(*8.计数器清零*)	
	IF GVL_State.iPLC_State=50 THEN
		(*-----------------------计数器清零操作-----------------------*)
		IF PLC_PRG.Step_Scout<=42 OR PLC_PRG.Step_Scout>=70 THEN
			iActNumPulse:=0;
			Entity_IO.bTriggerOut:=FALSE;
			Entity_IO.bTriggerPannel_NOT:=FALSE;
		END_IF
	ELSIF GVL_State.iPLC_State=60 THEN
		(*-----------------------计数器清零操作-----------------------*)
		IF PLC_PRG.Step_CBCT<=70 THEN
			iActNumPulse:=0;
			Entity_IO.bTriggerOut:=FALSE;
			Entity_IO.bTriggerPannel_NOT:=FALSE;
		END_IF
	ELSIF GVL_State.iPLC_State=40 THEN
		iActNumPulse:=0;
	END_IF

END_PROGRAM

// Device/Application/Motor
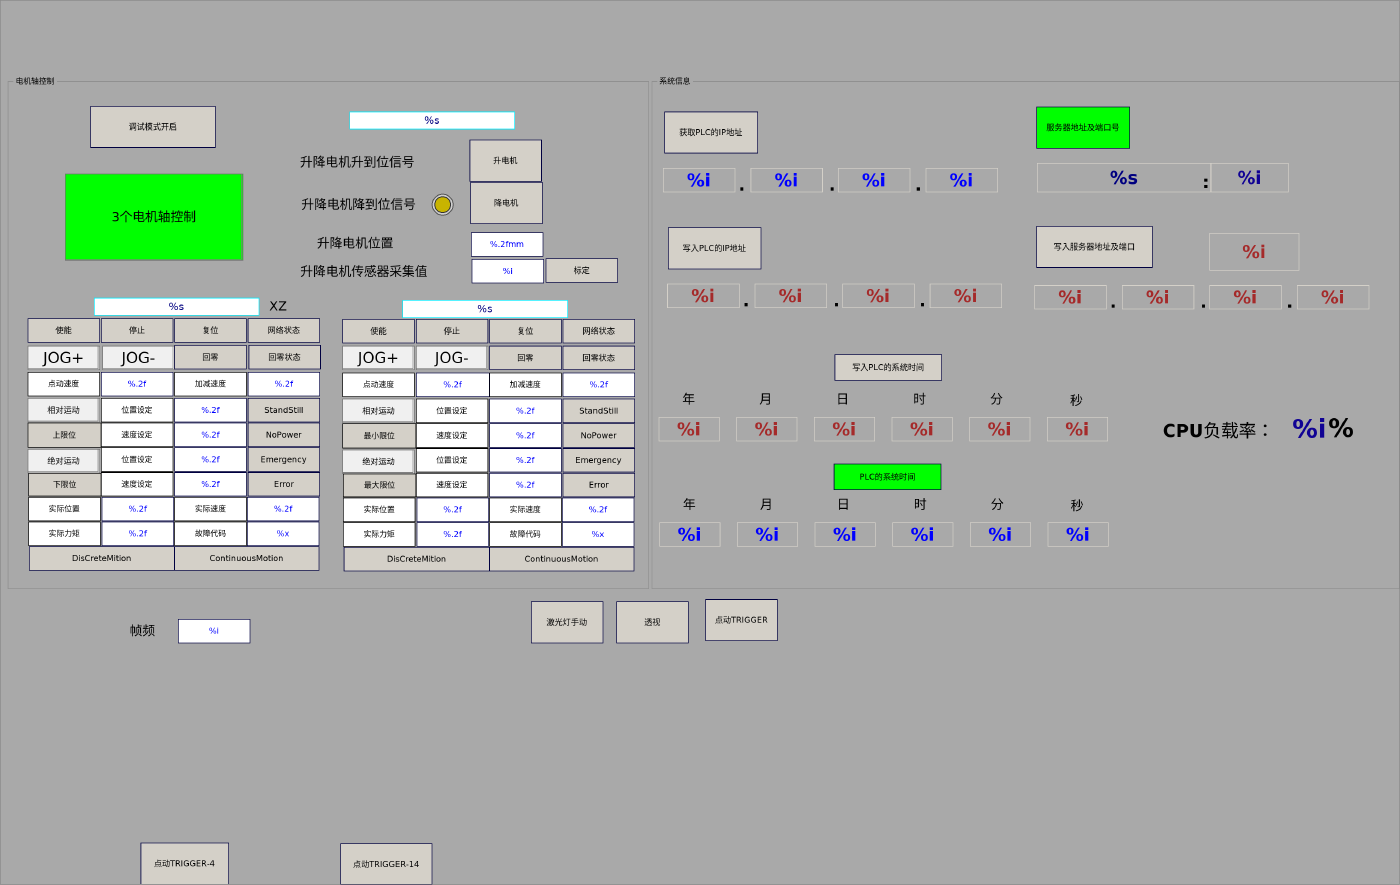
VISUALIZATION Motor  // 1983x1254
    Button (39,490 102x34), "JOG+", colour toggle: Axis_XZ.XZ_AxisCmd.bJogP
        tap Axis_XZ.XZ_AxisCmd.bJogP
    Rectangle (144,704 102x34), "%.2f", text variable: Axis_XZ.XZ_AxisState.rActPosition
    Button (145,490 102x34), "JOG-", colour toggle: Axis_XZ.XZ_AxisCmd.bJogN
        tap Axis_XZ.XZ_AxisCmd.bJogN
    RoundedRectangle (39,451 102x34), "使能", colour toggle: AXIS_XZ.XZ_AxisState.bPowering
        toggle Axis_XZ.XZ_AxisCmd.bPower
    RoundedRectangle (351,451 102x34), "网络状态", colour toggle: Axis_XZ.XZ_AxisState.bNetState
    Button (39,636 102x34), "绝对运动", colour toggle: Axis_XZ.XZ_AxisCmd.bAbs
        tap Axis_XZ.XZ_AxisCmd.bAbs
    Rectangle (40,704 102x34), "实际位置"
    Rectangle (350,704 102x34), "%.2f", text variable: Axis_XZ.XZ_AxisState.rActVelocity
    Rectangle (247,704 102x34), "实际速度"
    RoundedRectangle (143,451 102x34), "停止", colour toggle: Axis_XZ.XZ_AxisState.bStopState
        tap Axis_XZ.XZ_AxisCmd.bStop
    RoundedRectangle (247,451 102x34), "复位", colour toggle: Axis_XZ.XZ_AxisCmd.bReset
        tap Axis_XZ.XZ_AxisCmd.bReset
    Rectangle (133,422 234x25), "%s", text variable: InitMotor.sNameXZ, text list: ''
    Rectangle (247,739 102x34), "故障代码"
    Rectangle (350,739 102x34), "%x", text variable: Axis_XZ.XZ_AxisState.ErrorID, colour toggle: (Axis_XZ.XZ_AxisState.ErrorID)<>0
    Rectangle (40,670 103x33), "下限位", colour toggle: Entity_IO.bRotateMotorMax
    Rectangle (39,599 104x35), "上限位", colour toggle: Entity_IO.bRotateMotorMin
    RoundedRectangle (247,489 102x34), "回零", colour toggle: Axis_XZ.XZ_AxisCmd.bHome
        tap Axis_XZ.XZ_AxisCmd.bHome
    Button (39,564 102x34), "相对运动", colour toggle: Axis_XZ.XZ_AxisCmd.bRel
        tap Axis_XZ.XZ_AxisCmd.bRel
    Rectangle (143,527 102x34), "%.2f", text variable: Axis_XZ.XZ_AxisCmd.AxisPara.rJogVelocity
        OnMouseClick: write Axis_XZ.XZ_AxisCmd.AxisPara.rJogVelocity via Default
    Rectangle (39,527 102x34), "点动速度"
    Rectangle (247,527 102x34), "加减速度"
    Rectangle (351,527 102x34), "%.2f", text variable: Axis_XZ.XZ_AxisCmd.AxisPara.rAccDec
        OnMouseClick: write Axis_XZ.XZ_AxisCmd.AxisPara.rAccDec via Default
    Rectangle (143,564 102x34), "位置设定"
    Rectangle (247,564 102x34), "%.2f", text variable: Axis_XZ.XZ_AxisCmd.AxisPara.rRelPosition
        OnMouseClick: write Axis_XZ.XZ_AxisCmd.AxisPara.rRelPosition via Default
    Rectangle (143,599 102x34), "速度设定"
    Rectangle (247,599 102x34), "%.2f", text variable: Axis_XZ.XZ_AxisCmd.AxisPara.rRelVelocity
        OnMouseClick: write Axis_XZ.XZ_AxisCmd.AxisPara.rRelVelocity via Default
    Rectangle (143,634 102x34), "位置设定"
    Rectangle (693,635 102x34), "%.2f", text variable: Axis_QJ.QJ_AxisCmd.AxisPara.rAbsPosition
        OnMouseClick: write Axis_QJ.QJ_AxisCmd.AxisPara.rAbsPosition via Default
    Rectangle (143,669 102x34), "速度设定"
    Rectangle (247,669 102x34), "%.2f", text variable: Axis_XZ.XZ_AxisCmd.AxisPara.rAbsVelocity
        OnMouseClick: write Axis_XZ.XZ_AxisCmd.AxisPara.rAbsVelocity via Default
    RoundedRectangle (351,564 102x34), "StandStill", colour toggle: Axis_XZ.XZ_AxisState.bStandStill
    RoundedRectangle (351,599 102x34), "NoPower", colour toggle: Axis_XZ.XZ_AxisState.bPowerOff
    RoundedRectangle (351,634 102x34), "Emergency", colour toggle: Axis_XZ.XZ_AxisState.bErrStop
    RoundedRectangle (351,669 102x34), "Error", colour toggle: Axis_XZ.XZ_AxisState.bAxisErr
    Rectangle (144,739 102x34), "%.2f", text variable: Axis_XZ.XZ_AxisState.rActTorque
    Rectangle (40,739 102x34), "实际力矩"
    Rectangle (570,425 234x25), "%s", text variable: InitMotor.sNameQJ, text list: ''
    Button (485,490 102x34), "JOG+", colour toggle: Axis_QJ.QJ_AxisCmd.bJogP
        tap Axis_QJ.QJ_AxisCmd.bJogP
    Rectangle (590,705 102x34), "%.2f", text variable: Axis_QJ.QJ_AxisState.rActPosition
    Button (589,490 102x34), "JOG-", colour toggle: Axis_QJ.QJ_AxisCmd.bJogN
        tap Axis_QJ.QJ_AxisCmd.bJogN
    RoundedRectangle (485,452 102x34), "使能", colour toggle: AXIS_QJ.QJ_AxisState.bPowering
        toggle Axis_QJ.QJ_AxisCmd.bPower
    RoundedRectangle (797,452 102x34), "网络状态", colour toggle: Axis_QJ.QJ_AxisState.bNetState
    Button (485,637 102x34), "绝对运动", colour toggle: Axis_QJ.QJ_AxisCmd.bAbs
        tap Axis_QJ.QJ_AxisCmd.bAbs
    Rectangle (486,705 102x34), "实际位置"
    Rectangle (796,705 102x34), "%.2f", text variable: Axis_QJ.QJ_AxisState.rActVelocity
    Rectangle (693,705 102x34), "实际速度"
    RoundedRectangle (589,452 102x34), "停止", colour toggle: Axis_QJ.QJ_AxisCmd.bStop
        tap Axis_QJ.QJ_AxisCmd.bStop
    RoundedRectangle (693,452 102x34), "复位", colour toggle: Axis_QJ.QJ_AxisCmd.bReset
        tap Axis_QJ.QJ_AxisCmd.bReset
    Rectangle (693,740 102x34), "故障代码"
    Rectangle (796,740 102x34), "%x", text variable: Axis_QJ.QJ_AxisState.ErrorID, colour toggle: (Axis_QJ.QJ_AxisState.ErrorID)<>0
    Rectangle (486,671 103x33), "最大限位", colour toggle: Entity_IO.bForeMotorMax
    Rectangle (485,600 104x35), "最小限位", colour toggle: Entity_IO.bForeMotorMin
    RoundedRectangle (693,490 102x34), "回零", colour toggle: Axis_QJ.QJ_AxisCmd.bHome
        tap Axis_QJ.QJ_AxisCmd.bHome
    Button (485,565 102x34), "相对运动", colour toggle: Axis_QJ.QJ_AxisCmd.bRel
        tap Axis_QJ.QJ_AxisCmd.bRel
    Rectangle (589,528 104x34), "%.2f", text variable: Axis_QJ.QJ_AxisCmd.AxisPara.rJogVelocity
        OnMouseClick: write Axis_QJ.QJ_AxisCmd.AxisPara.rJogVelocity via Default
    Rectangle (485,528 102x34), "点动速度"
    Rectangle (693,528 102x34), "加减速度"
    Rectangle (797,528 102x34), "%.2f", text variable: Axis_QJ.QJ_AxisCmd.AxisPara.rAccDec
        OnMouseClick: write Axis_QJ.QJ_AxisCmd.AxisPara.rAccDec via Default
    Rectangle (589,565 102x34), "位置设定"
    Rectangle (693,565 102x34), "%.2f", text variable: Axis_QJ.QJ_AxisCmd.AxisPara.rRelPosition
        OnMouseClick: write Axis_QJ.QJ_AxisCmd.AxisPara.rRelPosition via Default, min -1000, max 1000
    Rectangle (589,600 102x34), "速度设定"
    Rectangle (693,600 102x34), "%.2f", text variable: Axis_QJ.QJ_AxisCmd.AxisPara.rRelVelocity
        OnMouseClick: write Axis_QJ.QJ_AxisCmd.AxisPara.rRelVelocity via Default
    Rectangle (589,635 102x34), "位置设定"
    Rectangle (247,634 102x34), "%.2f", text variable: Axis_XZ.XZ_AxisCmd.AxisPara.rAbsPosition
        OnMouseClick: write Axis_XZ.XZ_AxisCmd.AxisPara.rAbsPosition via Default
    Rectangle (589,670 102x34), "速度设定"
    Rectangle (693,670 102x34), "%.2f", text variable: Axis_QJ.QJ_AxisCmd.AxisPara.rAbsVelocity
        OnMouseClick: write Axis_QJ.QJ_AxisCmd.AxisPara.rAbsVelocity via Default
    RoundedRectangle (797,565 102x34), "StandStill", colour toggle: Axis_QJ.QJ_AxisState.bStandStill
    RoundedRectangle (797,600 102x34), "NoPower", colour toggle: Axis_QJ.QJ_AxisState.bPowerOff
    RoundedRectangle (797,635 102x34), "Emergency", colour toggle: Axis_QJ.QJ_AxisState.bErrStop
    RoundedRectangle (797,670 102x34), "Error", colour toggle: Axis_QJ.QJ_AxisState.bAxisErr
    Rectangle (590,740 102x34), "%.2f", text variable: Axis_QJ.QJ_AxisState.rActTorque
    Rectangle (486,740 102x34), "实际力矩"
    RoundedRectangle (487,775 206x34), "DisCreteMition", colour toggle: Axis_QJ.QJ_AxisState.bDisCreteMition
    RoundedRectangle (693,775 205x34), "ContinuousMotion", colour toggle: Axis_QJ.QJ_AxisState.bContinuousMotion
    RoundedRectangle (41,774 206x34), "DisCreteMition", colour toggle: Axis_XZ.XZ_AxisState.bDisCreteMition
    RoundedRectangle (247,774 205x34), "ContinuousMotion", colour toggle: Axis_XZ.XZ_AxisState.bContinuousMotion
    RoundedRectangle (128,150 177x59), "调试模式开启", colour toggle: WorkMode.bDebugMode
        toggle WorkMode.bDebugMode
    Rectangle (495,158 234x25), "%s", text variable: InitMotor.sNameSJ, text list: ''
    RoundedRectangle (665,198 102x59), "升电机", colour toggle: Entity_IO.bUpMotorPos
        tap Entity_IO.bUpMotorPos
    RoundedRectangle (666,258 102x59), "降电机", colour toggle: Entity_IO.bUpMotorNeg
        tap Entity_IO.bUpMotorNeg
    Label (410,212 192x36), "升降电机升到位信号"
    Label (412,272 192x36), "升降电机降到位信号"
    Lamp1 (608,272 38x36), variable: Entity_IO.bUpMotorMin, style: Lamp-Lamp1-Yellow
    Button (92,246 252x123), "3个电机轴控制"
        OnMouseClick:  Assign=Catalogue, Type=Assignment
    RoundedRectangle (773,366 102x34), "标定", colour toggle: Entity_IO.bCalibrate
        tap Entity_IO.bCalibrate
    Rectangle (667,329 102x34), "%.2fmm", text variable: Entity_IO.rRealPos
        OnMouseClick: write  via Default, min -100, max 1000
    Label (407,327 192x36), "升降电机位置"
    Rectangle (668,367 102x34), "%i", text variable: Entity_IO.AIX0
        OnMouseClick: write  via Default, min -100, max 1000
    Label (386,367 259x36), "升降电机传感器采集值"
    RoundedRectangle (352,489 102x34), "回零状态", colour toggle: Axis_XZ.XZ_AxisState.bHoming
    RoundedRectangle (797,490 102x34), "回零状态", colour toggle: Axis_QJ.QJ_AxisState.bHoming
    RoundedRectangle (941,158 132x59), "获取PLC的IP地址", colour toggle: PLC_PRG.bGetPLC_IP
        tap PLC_PRG.bGetPLC_IP
    Rectangle (939,238 102x34), "%i", text variable: PLC_PRG.LS_GetIPAddress_1.byIpSegmengt1
    Label (1033,248 36x26), "."
    Label (1161,248 36x26), "."
    Label (1283,248 36x26), "."
    Rectangle (1063,238 102x34), "%i", text variable: PLC_PRG.LS_GetIPAddress_1.byIpSegmengt2
    Rectangle (1187,238 102x34), "%i", text variable: PLC_PRG.LS_GetIPAddress_1.byIpSegmengt3
    Rectangle (1311,238 102x34), "%i", text variable: PLC_PRG.LS_GetIPAddress_1.byIpSegmengt4
    RoundedRectangle (946,322 132x59), "写入PLC的IP地址", colour toggle: PLC_PRG.bSetPLC_IP
        tap PLC_PRG.bSetPLC_IP
    Rectangle (945,402 102x34), "%i", text variable: PLC_PRG.LS_SetIPAddress_1.byIpSegmengt1
        OnMouseClick: write PLC_PRG.LS_SetIPAddress_1.byIpSegmengt1 via Default, min 0, max 1000
    Label (1039,412 36x26), "."
    Label (1167,412 36x26), "."
    Label (1289,412 36x26), "."
    Rectangle (1069,402 102x34), "%i", text variable: PLC_PRG.LS_SetIPAddress_1.byIpSegmengt2
        OnMouseClick: write PLC_PRG.LS_SetIPAddress_1.byIpSegmengt2 via Default, min 0, max 1000
    Rectangle (1193,402 102x34), "%i", text variable: PLC_PRG.LS_SetIPAddress_1.byIpSegmengt3
        OnMouseClick: write PLC_PRG.LS_SetIPAddress_1.byIpSegmengt3 via Default, min 0, max 1000
    Rectangle (1317,402 102x34), "%i", text variable: PLC_PRG.LS_SetIPAddress_1.byIpSegmengt4
        OnMouseClick: write PLC_PRG.LS_SetIPAddress_1.byIpSegmengt4 via Default, min 0, max 1000
    Rectangle (1817,583 76x49), "%i", text variable: PLC_PRG.rPLC_Load
    Label (1630,592 192x36), "CPU负载率："
    Label (1865,584 69x45), "%"
    Rectangle (933,591 86x34), "%i", text variable: PLC_PRG.LS_SetDintDT_1.uiYear
        OnMouseClick: write PLC_PRG.LS_SetDintDT_1.uiYear via Default, min 0, max 10000
    Rectangle (1043,591 86x34), "%i", text variable: PLC_PRG.LS_SetDintDT_1.uiMonth
        OnMouseClick: write PLC_PRG.LS_SetDintDT_1.uiMonth via Default, min 0, max 1000
    Rectangle (1153,591 86x34), "%i", text variable: PLC_PRG.LS_SetDintDT_1.uiDay
        OnMouseClick: write PLC_PRG.LS_SetDintDT_1.uiDay via Default, min 0, max 1000
    Rectangle (1263,591 86x34), "%i", text variable: PLC_PRG.LS_SetDintDT_1.uiHour
        OnMouseClick: write PLC_PRG.LS_SetDintDT_1.uiHour via Default, min 0, max 1000
    Rectangle (1373,591 86x34), "%i", text variable: PLC_PRG.LS_SetDintDT_1.uiMinute
        OnMouseClick: write PLC_PRG.LS_SetDintDT_1.uiMinute via Default, min 0, max 1000
    Rectangle (1483,591 86x34), "%i", text variable: PLC_PRG.LS_SetDintDT_1.uiSecond
        OnMouseClick: write PLC_PRG.LS_SetDintDT_1.uiSecond via Default, min 0, max 1000
    Label (942,548 67x36), "年"
    Label (1051,548 67x36), "月"
    Label (1160,548 67x36), "日"
    Label (1269,548 67x36), "时"
    Label (1378,548 67x36), "分"
    Label (1491,550 67x36), "秒"
    RoundedRectangle (1182,502 152x37), "写入PLC的系统时间", colour toggle: PLC_PRG.bSetSysTime
        tap PLC_PRG.bSetSysTime
    Rectangle (934,740 86x34), "%i", text variable: PLC_PRG.LS_ReadDintDT_1.uiYear
    Rectangle (1044,740 86x34), "%i", text variable: PLC_PRG.LS_ReadDintDT_1.uiMonth
    Rectangle (1154,740 86x34), "%i", text variable: PLC_PRG.LS_ReadDintDT_1.uiDay
    Rectangle (1264,740 86x34), "%i", text variable: PLC_PRG.LS_ReadDintDT_1.uiHour
    Rectangle (1374,740 86x34), "%i", text variable: PLC_PRG.LS_ReadDintDT_1.uiMinute
    Rectangle (1484,740 86x34), "%i", text variable: PLC_PRG.LS_ReadDintDT_1.uiSecond
    Label (943,697 67x36), "年"
    Label (1052,697 67x36), "月"
    Label (1161,697 67x36), "日"
    Label (1270,697 67x36), "时"
    Label (1379,697 67x36), "分"
    Label (1492,699 67x36), "秒"
    RoundedRectangle (1181,657 152x37), "PLC的系统时间"
    GroupBox (11,107 908x727), "电机轴控制"
        Label (287,309 192x36), "XZ"
    GroupBox (923,107 1060x727), "系统信息"
    Rectangle (1469,231 246x41), "%s", text variable: WorkStation_TCP.IP.sAddr, text list: ''
    Rectangle (1715,231 110x41), "%i", text variable: WorkStation_TCP.TCP_Client_1.uiPort
    Label (1685,239 46x37), ":"
    RoundedRectangle (1468,151 132x59), "服务器地址及端口号"
    RoundedRectangle (1468,320 164x59), "写入服务器地址及端口", colour toggle: WorkStation_TCP.bSetServerIP
        tap WorkStation_TCP.bSetServerIP
    Rectangle (1465,404 102x34), "%i", text variable: WorkStation_TCP.iServerIP1
        OnMouseClick: write WorkStation_TCP.iServerIP1 via Default, min 0, max 1000
    Label (1559,414 36x26), "."
    Label (1687,414 36x26), "."
    Label (1809,414 36x26), "."
    Rectangle (1589,404 102x34), "%i", text variable: WorkStation_TCP.iServerIP2
        OnMouseClick: write WorkStation_TCP.iServerIP2 via Default, min 0, max 1000
    Rectangle (1713,404 102x34), "%i", text variable: WorkStation_TCP.iServerIP3
        OnMouseClick: write WorkStation_TCP.iServerIP3 via Default, min 0, max 1000
    Rectangle (1837,404 102x34), "%i", text variable: WorkStation_TCP.iServerIP4
        OnMouseClick: write WorkStation_TCP.iServerIP4 via Default, min 0, max 1000
    Rectangle (1713,330 127x53), "%i", text variable: WorkStation_TCP.ServeruiPort
        OnMouseClick: write WorkStation_TCP.ServeruiPort via Default, min 0, max 65535
    RoundedRectangle (752,852 102x59), "激光灯手动", colour toggle: PLC_PRG.bDebug_Laser
        toggle PLC_PRG.bDebug_Laser
    RoundedRectangle (873,852 102x59), "透视", colour toggle: PLC_PRG.bTestXayOne
        toggle PLC_PRG.bTestXayOne
    RoundedRectangle (999,849 102x59), "点动TRIGGER", colour toggle: PLC_PRG.bTestTrigger
        tap PLC_PRG.bTestTrigger
    RoundedRectangle (199,1194 125x59), "点动TRIGGER-4", colour toggle: PLC_PRG.bTestTrigger11
        tap PLC_PRG.bTestTrigger11
    RoundedRectangle (482,1195 130x59), "点动TRIGGER-14", colour toggle: PLC_PRG.bTestTrigger22
        tap PLC_PRG.bTestTrigger22
    Rectangle (252,877 102x34), "%i", text variable: PLC_PRG.iSamplingRate1
        OnMouseClick: write PLC_PRG.iSamplingRate1 via Default, min 1, max 100000
    Label (109,876 185x36), "帧频"
END_VISUALIZATION

// Device/Application/Entity_IO
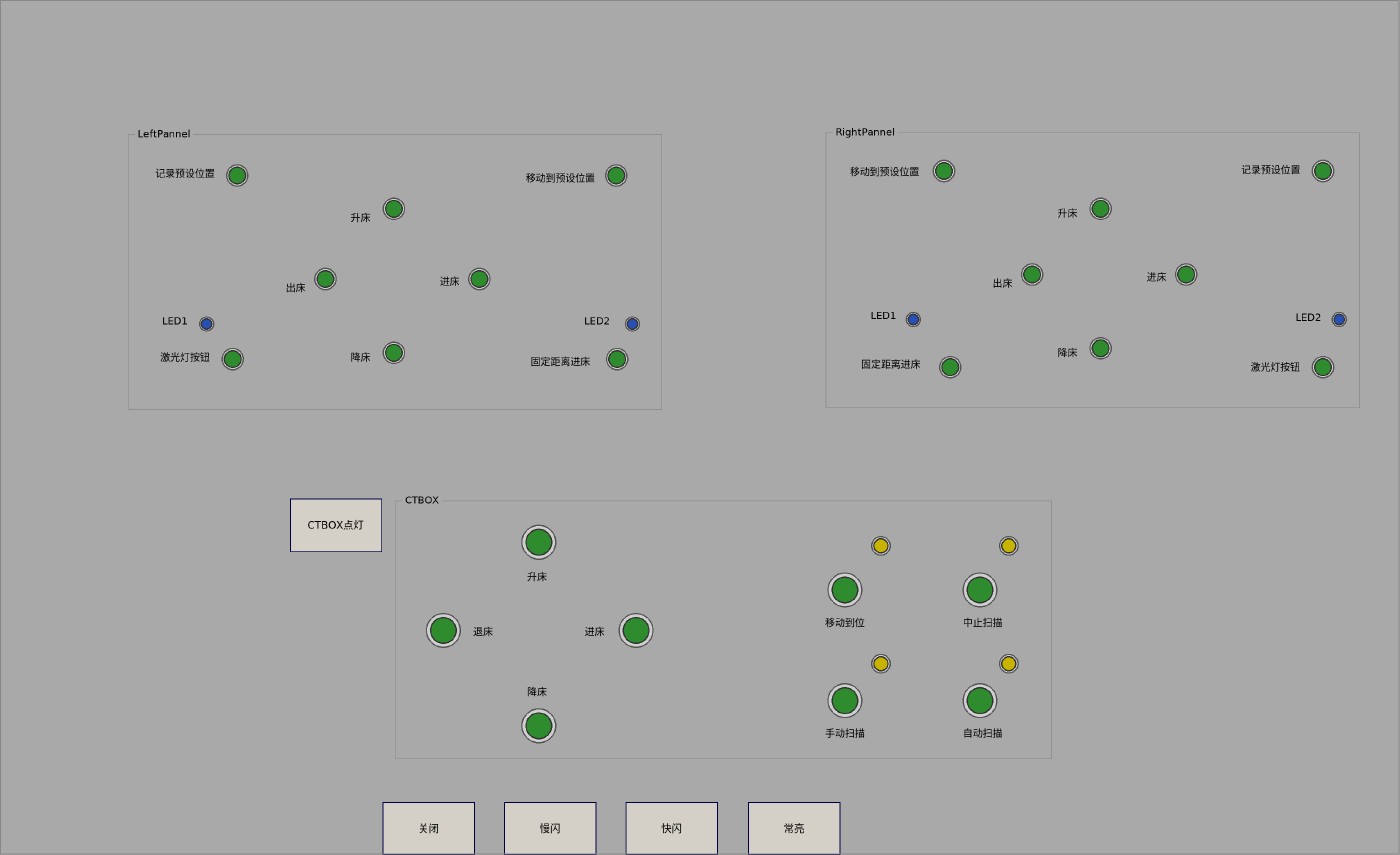
VISUALIZATION Entity_IO  // 1555x950
    Label (104,379 203x36), "激光灯按钮"
    Label (104,175 203x36), "记录预设位置"
    Lamp1 (423,217 29x30), variable: Entity_IO.LeftPannel_BedUp, style: Lamp-Lamp1-Green
    Lamp1 (423,377 29x30), variable: Entity_IO.LeftPannel_BedDown, style: Lamp-Lamp1-Green
    Label (299,379 203x36), "降床"
    Label (521,384 203x36), "固定距离进床"
    Label (227,302 203x36), "出床"
    Label (299,224 203x36), "升床"
    Label (398,295 203x36), "进床"
    Label (521,180 203x36), "移动到预设位置"
    Lamp1 (347,295 29x30), variable: Entity_IO.LeftPannel_BedBack, style: Lamp-Lamp1-Green
    Lamp1 (518,295 29x30), variable: Entity_IO.LeftPannel_BedFore, style: Lamp-Lamp1-Green
    Lamp1 (244,384 29x30), variable: Entity_IO.LeftPannel_LaserButton, style: Lamp-Lamp1-Green
    Lamp1 (249,180 29x30), variable: Entity_IO.LeftPannel_RecordPos, style: Lamp-Lamp1-Green
    Lamp1 (671,384 29x30), variable: Entity_IO.LeftPannel_DistanceMove, style: Lamp-Lamp1-Green
    Lamp1 (670,180 29x30), variable: Entity_IO.LeftPannel_MoveRecordPos, style: Lamp-Lamp1-Green
    Lamp1 (693,349 19x22), variable: Entity_IO.bLeftPannel_LED2, style: Lamp-Lamp1-Blue
    Lamp1 (220,349 19x22), variable: Entity_IO.bLeftPannel_LED1, style: Lamp-Lamp1-Blue
    Label (562,339 203x36), "LED2"
    Label (93,339 203x36), "LED1"
    Lamp1 (1208,372 29x30), variable: Entity_IO.RightPannel_BedDown, style: Lamp-Lamp1-Green
    Label (1084,374 203x36), "降床"
    Label (888,387 203x36), "固定距离进床"
    Label (1012,297 203x36), "出床"
    Label (1315,390 203x36), "激光灯按钮"
    Label (1310,171 203x36), "记录预设位置"
    Label (1084,219 203x36), "升床"
    Label (1183,290 203x36), "进床"
    Label (881,173 203x36), "移动到预设位置"
    Lamp1 (1132,290 29x30), variable: Entity_IO.RightPannel_BedBack, style: Lamp-Lamp1-Green
    Lamp1 (1303,290 29x30), variable: Entity_IO.RightPannel_BedFore, style: Lamp-Lamp1-Green
    Lamp1 (1455,393 29x30), variable: Entity_IO.RightPannel_LaserButton, style: Lamp-Lamp1-Green
    Lamp1 (1034,175 29x30), variable: Entity_IO.RightPannel_MoveRecordPos, style: Lamp-Lamp1-Green
    Lamp1 (1041,393 29x30), variable: Entity_IO.RightPannel_DistanceMove, style: Lamp-Lamp1-Green
    Lamp1 (1455,175 29x30), variable: Entity_IO.RightPannel_RecordPos, style: Lamp-Lamp1-Green
    Lamp1 (1478,344 19x22), variable: Entity_IO.bRightPannel_LED2, style: Lamp-Lamp1-Blue
    Lamp1 (1005,344 19x22), variable: Entity_IO.bRightPannel_LED1, style: Lamp-Lamp1-Blue
    Label (1352,335 203x36), "LED2"
    Label (880,333 203x36), "LED1"
    Lamp1 (1208,217 29x30), variable: Entity_IO.RightPannel_BedUp, style: Lamp-Lamp1-Green
    Lamp1 (576,580 45x45), variable: CTBOX_RS232.CTBOX_KEY[5], style: Lamp-Lamp1-Green
    Lamp1 (576,784 45x45), variable: CTBOX_RS232.CTBOX_KEY[7], style: Lamp-Lamp1-Green
    Lamp1 (684,678 45x45), variable: CTBOX_RS232.CTBOX_KEY[4], style: Lamp-Lamp1-Green
    Lamp1 (470,678 45x45), variable: CTBOX_RS232.CTBOX_KEY[6], style: Lamp-Lamp1-Green
    Lamp1 (916,633 45x45), variable: CTBOX_RS232.CTBOX_KEY[3], style: Lamp-Lamp1-Green
    Lamp1 (1066,633 45x45), variable: CTBOX_RS232.CTBOX_KEY[2], style: Lamp-Lamp1-Green
    Lamp1 (916,756 45x45), variable: CTBOX_RS232.CTBOX_KEY[0], style: Lamp-Lamp1-Green
    Lamp1 (1066,756 45x45), variable: CTBOX_RS232.CTBOX_KEY[1], style: Lamp-Lamp1-Green
    Lamp1 (966,725 25x25), variable: CTBOX_RS232.Lamp7State<>0, style: Lamp-Lamp1-Yellow
    Lamp1 (1108,725 25x25), variable: CTBOX_RS232.Lamp8State<>0, style: Lamp-Lamp1-Yellow
    Lamp1 (966,594 25x25), variable: CTBOX_RS232.Lamp5State<>0, style: Lamp-Lamp1-Yellow
    Lamp1 (1108,594 25x25), variable: CTBOX_RS232.Lamp6State<>0, style: Lamp-Lamp1-Yellow
    GroupBox (142,141 593x314), "LeftPannel"
    GroupBox (917,139 593x314), "RightPannel"
    GroupBox (439,548 729x295), "CTBOX"
    Label (515,623 163x36), "升床"
    Label (515,751 163x36), "降床"
    Label (455,684 163x36), "退床"
    Label (579,684 163x36), "进床"
    Label (857,674 163x36), "移动到位"
    Label (1010,674 163x36), "中止扫描"
    Label (857,797 163x36), "手动扫描"
    Label (1010,797 163x36), "自动扫描"
    RoundedRectangle (322,554 102x59), "CTBOX点灯", colour toggle: CTBOX_RS232.bDebug_RS232
        toggle CTBOX_RS232.bDebug_RS232
    RoundedRectangle (425,891 102x59), "关闭", colour toggle: CTBOX_RS232.A1
        toggle CTBOX_RS232.A1
    RoundedRectangle (560,891 102x59), "慢闪", colour toggle: CTBOX_RS232.A2
        toggle CTBOX_RS232.A2
    RoundedRectangle (695,891 102x59), "快闪", colour toggle: CTBOX_RS232.A3
        toggle CTBOX_RS232.A3
    RoundedRectangle (831,891 102x59), "常亮", colour toggle: CTBOX_RS232.A4
        toggle CTBOX_RS232.A4
END_VISUALIZATION
